// Mitsubishi GX Works2 project: 모터5   PLC: Q02/Q02H

PROGRAM MAIN
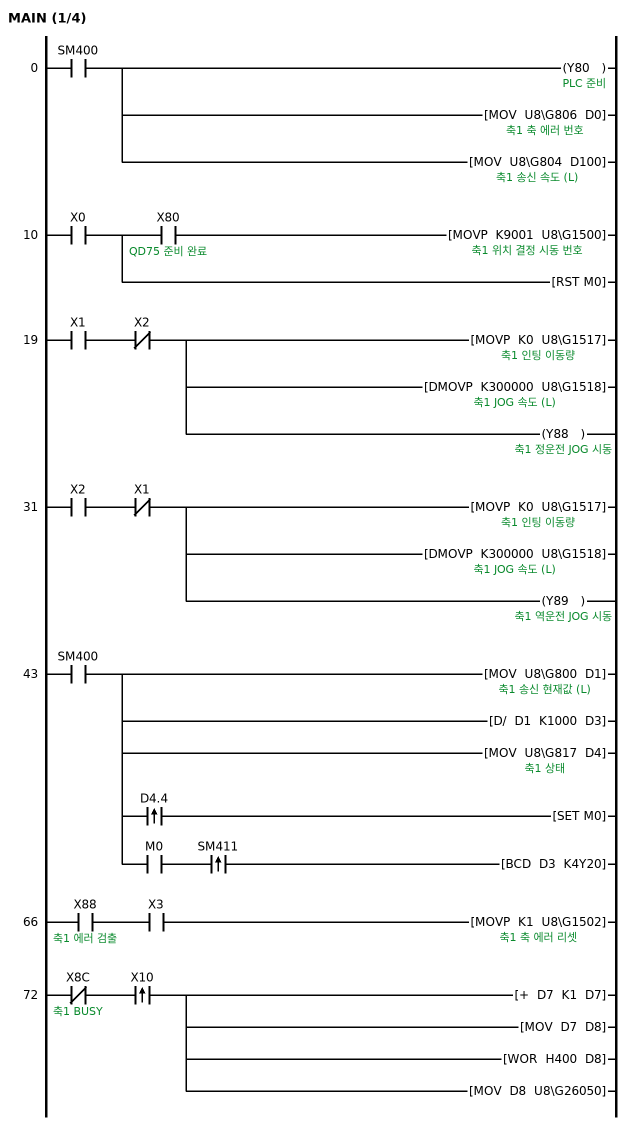
0     LD      SM400
      OUT     Y80  ; PLC 준비
      MOV     U8\G806 D0  ; 축1 축 에러 번호
      MOV     U8\G804 D100  ; 축1 송신 속도 (L)
10    LD      X0
      MPS
      AND     X80  ; QD75 준비 완료
      MOVP    K9001 U8\G1500  ; 축1 위치 결정 시동 번호
      MPP
      RST     M0
19    LD      X1
      ANI     X2
      MOVP    K0 U8\G1517  ; 축1 인팅 이동량
      DMOVP   K300000 U8\G1518  ; 축1 JOG 속도 (L)
      OUT     Y88  ; 축1 정운전 JOG 시동
31    LD      X2
      ANI     X1
      MOVP    K0 U8\G1517
      DMOVP   K300000 U8\G1518
      OUT     Y89  ; 축1 역운전 JOG 시동
43    LD      SM400
      MOV     U8\G800 D1  ; 축1 송신 현재값 (L)
      D/      D1 K1000 D3
      MOV     U8\G817 D4  ; 축1 상태
      MPS
      ANDP    D4.4
      SET     M0
      MPP
      AND     M0
      ANDP    SM411
      BCD     D3 K4Y20
66    LD      X88  ; 축1 에러 검출
      AND     X3
      MOVP    K1 U8\G1502  ; 축1 축 에러 리셋
72    LDI     X8C  ; 축1 BUSY
      ANDP    X10
      +       D7 K1 D7
      MOV     D7 D8
      WOR     H400 D8
      MOV     D8 U8\G26050
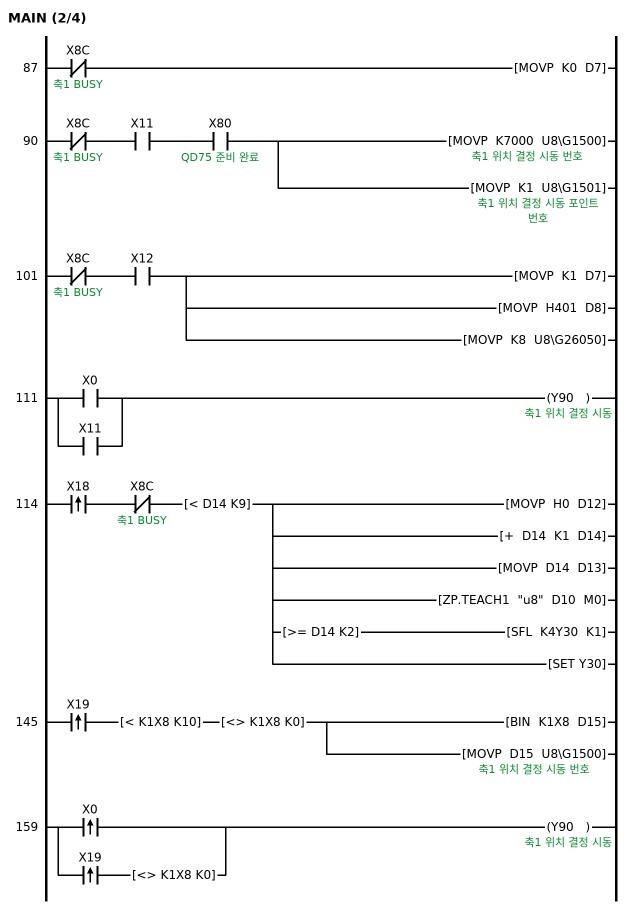
87    LDI     X8C  ; 축1 BUSY
      MOVP    K0 D7
90    LDI     X8C  ; 축1 BUSY
      AND     X11
      AND     X80  ; QD75 준비 완료
      MOVP    K7000 U8\G1500
      MOVP    K1 U8\G1501  ; 축1 위치 결정 시동 포인트 번호
101   LDI     X8C  ; 축1 BUSY
      AND     X12
      MOVP    K1 D7
      MOVP    H401 D8
      MOVP    K8 U8\G26050
111   LD      X0
      OR      X11
      OUT     Y90  ; 축1 위치 결정 시동
114   LDP     X18
      ANI     X8C  ; 축1 BUSY
      AND<    D14 K9
      MOVP    H0 D12
      +       D14 K1 D14
      MOVP    D14 D13
      ZP.TEACH1 "u8" D10 M0
      MPS
      AND>=   D14 K2
      SFL     K4Y30 K1
      MPP
      SET     Y30
145   LDP     X19
      AND<    K1X8 K10
      AND<>   K1X8 K0
      BIN     K1X8 D15
      MOVP    D15 U8\G1500
159   LDP     X0
      LDP     X19
      AND<>   K1X8 K0
      ORB
      OUT     Y90  ; 축1 위치 결정 시동
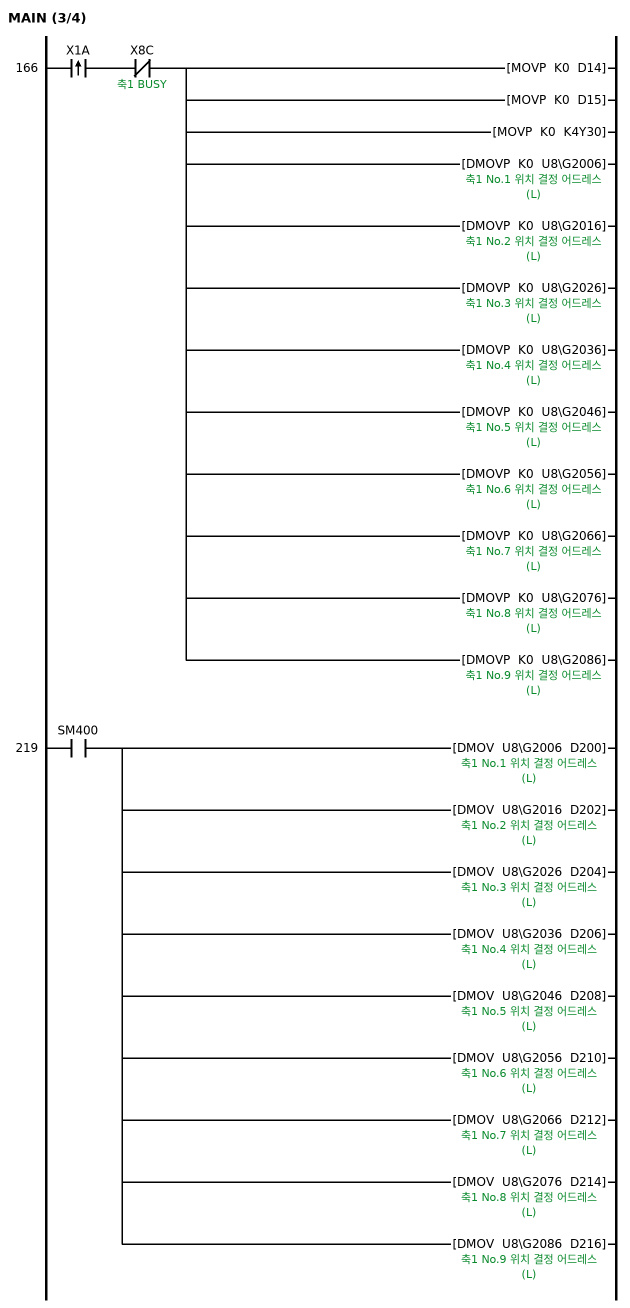
166   LDP     X1A
      ANI     X8C  ; 축1 BUSY
      MOVP    K0 D14
      MOVP    K0 D15
      MOVP    K0 K4Y30
      DMOVP   K0 U8\G2006  ; 축1 No.1 위치 결정 어드레스 (L)
      DMOVP   K0 U8\G2016  ; 축1 No.2 위치 결정 어드레스 (L)
      DMOVP   K0 U8\G2026  ; 축1 No.3 위치 결정 어드레스 (L)
      DMOVP   K0 U8\G2036  ; 축1 No.4 위치 결정 어드레스 (L)
      DMOVP   K0 U8\G2046  ; 축1 No.5 위치 결정 어드레스 (L)
      DMOVP   K0 U8\G2056  ; 축1 No.6 위치 결정 어드레스 (L)
      DMOVP   K0 U8\G2066  ; 축1 No.7 위치 결정 어드레스 (L)
      DMOVP   K0 U8\G2076  ; 축1 No.8 위치 결정 어드레스 (L)
      DMOVP   K0 U8\G2086  ; 축1 No.9 위치 결정 어드레스 (L)
219   LD      SM400
      DMOV    U8\G2006 D200
      DMOV    U8\G2016 D202
      DMOV    U8\G2026 D204
      DMOV    U8\G2036 D206
      DMOV    U8\G2046 D208
      DMOV    U8\G2056 D210
      DMOV    U8\G2066 D212
      DMOV    U8\G2076 D214
      DMOV    U8\G2086 D216
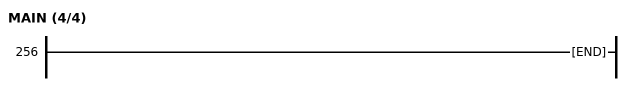
256   END
END_PROGRAM

// device comments not shown above
X81  ; 동기용 플래그
X84  ; 축1 M 코드 ON
X85  ; 축2 M 코드 ON
X89  ; 축2 에러 검출
X8D  ; 축2 BUSY
X90  ; 축1 시동 완료
X91  ; 축2 시동 완료
X94  ; 축1 위치 결정 완료
X95  ; 축2 위치 결정 완료
Y84  ; 축1 축 정지
Y85  ; 축2 축 정지
Y8A  ; 축2 정운전 JOG 시동
Y8B  ; 축2 역운전 JOG 시동
Y91  ; 축2 위치 결정 시동
Y94  ; 축1 실행 금지 플래그
Y95  ; 축2 실행 금지 플래그
